SUBAPPLICATION Uebung_016 (* Background Colour umschalten *)
  (* Standard: 61499-2; Description: Copyright (c) 2023 Meisterschulen am Ostbahnhof This program and the accompanying materials are made available under the terms of the Eclipse Public License 2.0 which is available at https://www.eclipse.org/legal/epl-2.0/ SPDX-License-Identifier: EPL-2.0 *)
  (* Version 1.0, 2023-10-23, Franz Höpfinger, Meisterschulen am Ostbahnhof *)
  PACKAGE Uebungen;
  IMPORT isobus::UT::io::Softkey::SoftKeyActivationCode::SK_RELEASED;
  IMPORT Uebungen::const::UT::DefaultPool::SoftKey_F1;
  IMPORT Uebungen::const::UT::DefaultPool::SoftKey_F2;
  IMPORT Uebungen::const::UT::DefaultPool::SoftKey_F7;
  IMPORT isobus::UT::Q::colours::COLOR_GREEN;
  IMPORT isobus::UT::Q::colours::COLOR_WHITE;
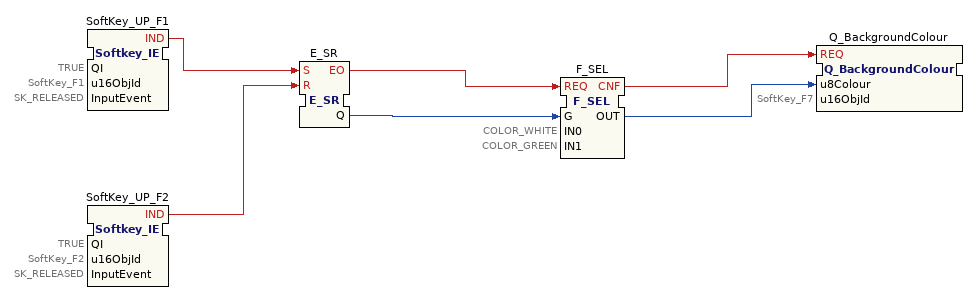
  FBS
    SoftKey_UP_F1 : isobus::UT::io::Softkey::Softkey_IE(QI := TRUE, u16ObjId := SoftKey_F1, InputEvent := SK_RELEASED);
    SoftKey_UP_F2 : isobus::UT::io::Softkey::Softkey_IE(QI := TRUE, u16ObjId := SoftKey_F2, InputEvent := SK_RELEASED);
    E_SR : iec61499::events::E_SR;
    F_SEL : iec61131::selection::F_SEL(IN0 := COLOR_WHITE, IN1 := COLOR_GREEN);
    Q_BackgroundColour : isobus::UT::Q::Q_BackgroundColour(u16ObjId := SoftKey_F7);
  END_FBS
  EVENT_CONNECTIONS
    SoftKey_UP_F1.IND TO E_SR.S;
    SoftKey_UP_F2.IND TO E_SR.R;
    E_SR.EO TO F_SEL.REQ;
    F_SEL.CNF TO Q_BackgroundColour.REQ;
  END_CONNECTIONS
  DATA_CONNECTIONS
    E_SR.Q TO F_SEL.G;
    F_SEL.OUT TO Q_BackgroundColour.u8Colour;
  END_CONNECTIONS
END_SUBAPPLICATION
